FUNCTION_BLOCK StateManager
VAR_IN_OUT
	statelist: ARRAY[*] OF IState;
END_VAR
VAR
	index: INT:=1;
	message: String;
END_VAR

METHOD RunProcess : BOOL
IF THIS^.statelist[index]<>0 THEN
	IF THIS^.statelist[index].execute() THEN
		IF index<= SIZEOF(statelist)-1 THEN		
			index:=index+1;
		ELSE
			index:=1;
		END_IF
	END_IF
	message:= THIS^.statelist[index].Description;
END_IF
END_METHOD

END_FUNCTION_BLOCK

(* stored: Version 1.1.0.1
   POU StateManager: Id {cd44a106-8778-4274-94ba-bd71d7d0087f}, SpecialFunc None
   Method RunProcess: Id {71358e19-649b-4bb9-8fbc-912ca4112b8e} *)
